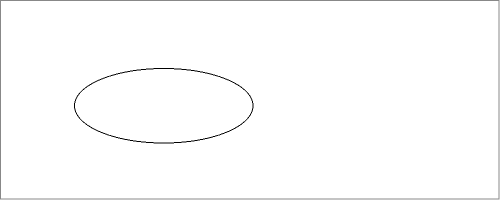
VISUALIZATION DialogTimer  // 500x200
    Ellipse (74,68 179x75)
END_VISUALIZATION

(* stored: Version 1.1.0.1, ProductVersion 3.1.4024.3
   Visu DialogTimer: Id {7b51e6c6-1e03-4e25-8b27-34dbdd270a32} *)
